ABB RAPID module: MainModule.mod

MODULE MainModule

    PERS robtarget POSITIONS0{30}:=[[[-127,-642,417],[0.0841205,-0.0345642,-0.628484,0.772488],[-2,-1,-2,1],[9E+9,9E+9,9E+9,9E+9,9E+9,9E+9]],
        [[-147,-644.16,415.65],[0.106262,-0.0312222,-0.640695,0.759766],[-2,-1,-2,1],[9E+9,9E+9,9E+9,9E+9,9E+9,9E+9]],
                [[275.78,-364.53,870.93],[0.0855649,-0.355297,0.349162,-0.862861],[-1,-1,-2,1],[9E+9,9E+9,9E+9,9E+9,9E+9,9E+9]],
                        [[275.78,-364.53,870.93],[0.0855649,-0.355297,0.349162,-0.862861],[-1,-1,-2,1],[9E+9,9E+9,9E+9,9E+9,9E+9,9E+9]],
                                [[275.78,-364.53,870.93],[0.0855649,-0.355297,0.349162,-0.862861],[-1,-1,-2,1],[9E+9,9E+9,9E+9,9E+9,9E+9,9E+9]],
                                        [[275.78,-364.53,870.93],[0.0855897,-0.35532,0.349124,-0.862864],[-1,-1,-2,1],[9E+9,9E+9,9E+9,9E+9,9E+9,9E+9]],
                                                [[275.78,-364.53,870.93],[0.0855897,-0.35532,0.349124,-0.862864],[-1,-1,-2,1],[9E+9,9E+9,9E+9,9E+9,9E+9,9E+9]],
                                                        [[275.78,-364.53,870.93],[0.0855897,-0.35532,0.349124,-0.862864],[-1,-1,-2,1],[9E+9,9E+9,9E+9,9E+9,9E+9,9E+9]],
                                                                [[275.78,-364.53,870.93],[0.0855897,-0.35532,0.349124,-0.862864],[-1,-1,-2,1],[9E+9,9E+9,9E+9,9E+9,9E+9,9E+9]],
                                                                        [[275.78,-364.53,870.93],[0.0855897,-0.35532,0.349124,-0.862864],[-1,-1,-2,1],[9E+9,9E+9,9E+9,9E+9,9E+9,9E+9]],
                                                                                [[275.78,-364.53,870.93],[0.0855897,-0.35532,0.349124,-0.862864],[-1,-1,-2,1],[9E+9,9E+9,9E+9,9E+9,9E+9,9E+9]],
                                                                                        [[275.78,-364.53,870.93],[0.0855897,-0.35532,0.349124,-0.862864],[-1,-1,-2,1],[9E+9,9E+9,9E+9,9E+9,9E+9,9E+9]],
                                                                                                [[275.78,-364.53,870.93],[0.0855897,-0.35532,0.349124,-0.862864],[-1,-1,-2,1],[9E+9,9E+9,9E+9,9E+9,9E+9,9E+9]],
        [[275.78,-364.53,870.93],[0.0855897,-0.35532,0.349124,-0.862864],[-1,-1,-2,1],[9E+9,9E+9,9E+9,9E+9,9E+9,9E+9]],
                [[275.78,-364.53,870.93],[0.0855897,-0.35532,0.349124,-0.862864],[-1,-1,-2,1],[9E+9,9E+9,9E+9,9E+9,9E+9,9E+9]],
                        [[275.78,-364.53,870.93],[0.0855897,-0.35532,0.349124,-0.862864],[-1,-1,-2,1],[9E+9,9E+9,9E+9,9E+9,9E+9,9E+9]],
                                [[275.78,-364.53,870.93],[0.0855897,-0.35532,0.349124,-0.862864],[-1,-1,-2,1],[9E+9,9E+9,9E+9,9E+9,9E+9,9E+9]],
        [[275.78,-364.53,870.93],[0.0855897,-0.35532,0.349124,-0.862864],[-1,-1,-2,1],[9E+9,9E+9,9E+9,9E+9,9E+9,9E+9]],
                [[275.78,-364.53,870.93],[0.0855897,-0.35532,0.349124,-0.862864],[-1,-1,-2,1],[9E+9,9E+9,9E+9,9E+9,9E+9,9E+9]],
                        [[275.78,-364.53,870.93],[0.0855897,-0.35532,0.349124,-0.862864],[-1,-1,-2,1],[9E+9,9E+9,9E+9,9E+9,9E+9,9E+9]],
                                [[275.78,-364.53,870.93],[0.0855897,-0.35532,0.349124,-0.862864],[-1,-1,-2,1],[9E+9,9E+9,9E+9,9E+9,9E+9,9E+9]],
                                        [[275.78,-364.53,870.93],[0.0855897,-0.35532,0.349124,-0.862864],[-1,-1,-2,1],[9E+9,9E+9,9E+9,9E+9,9E+9,9E+9]],
                                                [[275.78,-364.53,870.93],[0.0855897,-0.35532,0.349124,-0.862864],[-1,-1,-2,1],[9E+9,9E+9,9E+9,9E+9,9E+9,9E+9]],
                                                        [[275.78,-364.53,870.93],[0.0855897,-0.35532,0.349124,-0.862864],[-1,-1,-2,1],[9E+9,9E+9,9E+9,9E+9,9E+9,9E+9]],

                                                                [[275.78,-364.53,870.93],[0.0855897,-0.35532,0.349124,-0.862864],[-1,-1,-2,1],[9E+9,9E+9,9E+9,9E+9,9E+9,9E+9]],
                                                                            [[275.78,-364.53,870.93],[0.0855897,-0.35532,0.349124,-0.862864],[-1,-1,-2,1],[9E+9,9E+9,9E+9,9E+9,9E+9,9E+9]],
                                                                                    [[275.78,-364.53,870.93],[0.0855897,-0.35532,0.349124,-0.862864],[-1,-1,-2,1],[9E+9,9E+9,9E+9,9E+9,9E+9,9E+9]],
                                                                                            [[275.78,-364.53,870.93],[0.0855897,-0.35532,0.349124,-0.862864],[-1,-1,-2,1],[9E+9,9E+9,9E+9,9E+9,9E+9,9E+9]],
                                        [[275.78,-364.53,870.93],[0.0855897,-0.35532,0.349124,-0.862864],[-1,-1,-2,1],[9E+9,9E+9,9E+9,9E+9,9E+9,9E+9]],
                                                                                                        [[275.78,-364.53,870.93],[0.0855897,-0.35532,0.349124,-0.862864],[-1,-1,-2,1],[9E+9,9E+9,9E+9,9E+9,9E+9,9E+9]]
        ];
    !PERS robtarget POSITIONS0{50};
    PERS dnum Float32s0{500};
    PERS dnum Int32s0{500};
    PERS bool WRs0{500};

    PROC main()
        WRs0{1}:=NOT WRs0{1};
        Int32s0{1}:=Int32s0{1}+1;
        Float32s0{1}:=Float32s0{1}+1.3;
        MoveJ POSITIONS0{1},v1000,z50,tool0;
        MoveJ POSITIONS0{2},v1000,z50,tool0;
        MoveJ POSITIONS0{1},v1000,z50,tool0;
    ENDPROC
ENDMODULE
